// TIA Portal V18 export
DATA_BLOCK "DB"   // DB1
{ S7_Optimized_Access := 'TRUE' }
VERSION : 0.1
// stored: AutoNumber true, DBAccessibleFromOPCUA true, DBAccessibleFromWebserver true, IsOnlyStoredInLoadMemory false, IsRetainMemResEnabled false, IsWriteProtectedInAS false, MemoryReserve 100
   VAR
      ON : Bool;
      OFF : Bool;
      LAMP : Bool;
      ERROR : Bool;
      STATUS : Word;
      BPOWER : Bool;
   END_VAR
BEGIN
END_DATA_BLOCK
